FUNCTION_BLOCK FB_MessageBuffer
VAR
	fbMemRingBuffer : FB_MemRingBuffer;
	BufferArray  : ARRAY [0..100] OF BYTE;
END_VAR

METHOD PUBLIC AddMessage
VAR_INPUT
	eMessage : REFERENCE TO STRING;
END_VAR
fbMemRingBuffer.A_AddTail(	pWrite := ADR(eMessage),
							cbWrite := SIZEOF(eMessage),
							pBuffer := ADR(BufferArray),
							cbBuffer := SIZEOF(BufferArray));
END_METHOD

METHOD PUBLIC GetAndRemoveMessage
VAR_OUTPUT
	eMessage : STRING;
END_VAR
fbMemRingBuffer.A_RemoveHead(	pRead := ADR(eMessage),
								cbRead := SIZEOF(eMessage),
								pBuffer := ADR(BufferArray),
								cbBuffer := SIZEOF(BufferArray));
END_METHOD

PROPERTY PUBLIC getNumberOfMessages : UDINT
GET
getNumberOfMessages := fbMemRingBuffer.nCount;
END_GET
END_PROPERTY

END_FUNCTION_BLOCK

(* stored: Version 1.1.0.1, ProductVersion 3.1.4024.12
   POU FB_MessageBuffer: Id {19c240da-5dca-4c00-9805-e99bbf7dd140}, SpecialFunc None
   Method AddMessage: Id {10861b0c-e4dc-4f76-ad1b-444150214bee}
   Method GetAndRemoveMessage: Id {22f69b0d-8347-4238-ac95-590cf2cb5e32}
   Property getNumberOfMessages: Id {d73ba38a-c184-40d5-91be-9787bdda7d25}
   Get Get: Id {31fe221b-da92-45e7-a96e-0b5402f9b0d0} *)
